// TwinCAT 3 PLC project ASRS
// ProgramVersion: 3.1.4024.0
// libraries:
//   Tc2_Standard, * (Beckhoff Automation GmbH)
//   Tc2_System, * (Beckhoff Automation GmbH)
//   Tc3_Module, * (Beckhoff Automation GmbH)
// project tree:
//   / Class Diagram.TcCD (not stored), Class Diagram_1.TcCD (not stored), PlcTask.TcTTO
//   DUTs/Enum/ E_ConveyorMode.TcDUT, E_DiverterState.TcDUT, E_CraneState.TcDUT, E_AisleMode.TcDUT, E_SlotStatus.TcDUT, E_WarehouseState.TcDUT
//   DUTs/Structure/ ST_Alarm.TcDUT, ST_Parcel.TcDUT, ST_StorageSlot.TcDUT, ST_Position.TcDUT, ST_CraneJob.TcDUT, ST_HMI_Search.TcDUT (not stored)
//   GVLs/ GVL_IO.TcGVL, GVL_Config.TcGVL, GVL_Warehouse.TcGVL
//   POUs/ITFs/ I_Conveyor.TcIO, I_Diverter.TcIO, I_Crane.TcIO
//   POUs/Entity/ FB_Conveyor.TcPOU, FB_BiDirectionConveyor.TcPOU, FB_RAT.TcPOU, FB_Crane.TcPOU
//   POUs/Controller/ FB_InFeedController.TcPOU, FB_LoopController.TcPOU, FB_AisleController.TcPOU, FB_CraneController.TcPOU, FB_OutFeedController.TcPOU
//   POUs/ FB_WareHouseController.TcPOU, MAIN.TcPOU
// real-time tasks:
//   TASK PlcTask: cycle T#10ms, priority 20, ADS port 350
//   TASK PlcTask1: cycle T#10ms, priority 21, ADS port 351

CONFIGURATION ASRS
    RESOURCE PLC ON TwinCAT3
        TASK PlcTask(INTERVAL := T#10ms, PRIORITY := 20);
        PROGRAM MAIN WITH PlcTask : MAIN;
    END_RESOURCE
END_CONFIGURATION

// ---- DUTs/Enum/E_ConveyorMode.TcDUT
{attribute 'qualified_only'}
{attribute 'strict'}

TYPE E_ConveyorMode :
(
    IDLE              := 0,
    RUNNING_FORWARD   := 1,
    RUNNING_BACKWARD  := 2,
    FAULT             := 3
);
END_TYPE

// ---- DUTs/Enum/E_DiverterState.TcDUT
{attribute 'qualified_only'}
{attribute 'strict'}
{attribute 'reflection'}
TYPE E_DiverterState :
(
    IDLE      := 0,
    LIFTING   := 10,
    DIVERTING := 20,
    LOWERING  := 30,
	DONE := 40,
    FAULT     := 90
);
END_TYPE

// ---- DUTs/Enum/E_CraneState.TcDUT
{attribute 'qualified_only'}
{attribute 'strict'}
TYPE E_CraneState :
(
    IDLE            := 0,
    MOVING_TO_PICK  := 10,
	READY_TO_PICK   := 15,
    PICKING         := 20,
	READY_TO_MOVE   := 25,
    MOVING_TO_PLACE := 30,
    PLACING         := 40,
    RETURNING_HOME  := 50,
    FAULT           := 99
);
END_TYPE

// ---- DUTs/Enum/E_AisleMode.TcDUT
{attribute 'qualified_only'}
{attribute 'strict'}
TYPE E_AisleMode :
(
    IDLE                := 0,
    RECEIVING_FROM_LOOP := 10,
    TRANSPORT_TO_CRANE  := 20,
    WAITING_FOR_PICK    := 30,
    READY_FOR_DROP      := 40,
    TRANSPORT_TO_LOOP   := 50,
    FAULT               := 99
);
END_TYPE

// ---- DUTs/Enum/E_SlotStatus.TcDUT
{attribute 'qualified_only'}
{attribute 'strict'}
TYPE E_SlotStatus :
(
    EMPTY        := 0,
    RESERVED_IN  := 1,
    OCCUPIED     := 2,
    RESERVED_OUT := 3,
    BLOCKED      := 4
);
END_TYPE

// ---- DUTs/Enum/E_WarehouseState.TcDUT
{attribute 'qualified_only'}
{attribute 'strict'}
TYPE E_WarehouseState :
(
    IDLE    := 0,
    RUNNING := 1,
    PAUSED  := 2,
    FAULT   := 99
);
END_TYPE

// ---- DUTs/Structure/ST_Alarm.TcDUT
TYPE ST_Alarm :
STRUCT
	bActive     : BOOL;
    sSource     : STRING(50);
    sMessage    : STRING(100);
END_STRUCT
END_TYPE

// ---- DUTs/Structure/ST_Parcel.TcDUT
TYPE ST_Parcel :
STRUCT
    sID          : STRING(20);
    sDescription : STRING(40);
    fWeight      : REAL;
    nTargetAisle : INT;
    bIsHeavy     : BOOL;
END_STRUCT
END_TYPE

// ---- DUTs/Structure/ST_StorageSlot.TcDUT
TYPE ST_StorageSlot :
STRUCT
    eStatus      : E_SlotStatus;
    stParcel     : ST_Parcel;
    bIsRear      : BOOL;
    bMaintenance : BOOL;
END_STRUCT
END_TYPE

// ---- DUTs/Structure/ST_Position.TcDUT
TYPE ST_Position :
STRUCT
    nCol            : INT;
    nRow            : INT;
    fTargetX        : LREAL;
    fTargetY        : LREAL;
    bIsAisleStation : BOOL;
END_STRUCT
END_TYPE

// ---- DUTs/Structure/ST_CraneJob.TcDUT
TYPE ST_CraneJob :
STRUCT
    bValid    : BOOL;
    bIsStore  : BOOL;
    nAisle    : INT;
    stRackPos : ST_Position;
    stParcel  : ST_Parcel;
END_STRUCT
END_TYPE

// ---- GVLs/GVL_IO.TcGVL
{attribute 'qualified_only'}
VAR_GLOBAL
	

	bParcelReady            : BOOL;
	bOutfeedReq             : BOOL;
    // Infeed conveyor
    bInfeedSensor           : BOOL;
    bInfeedBlocker          : BOOL;
    bInfeedMotor            : BOOL;

    // Infeed RAT (transfers parcel from infeed conveyor onto loop)
    bInfeedRatSensor        : BOOL;
    bInfeedRatLift          : BOOL;
    bInfeedRatTravel        : BOOL;
    bInfeedRatUp            : BOOL;
    bInfeedRatDown          : BOOL;

    // Main loop conveyor
    bLoopMotor              : BOOL;
    bLoopSensor             : BOOL;
	bLoopParcelMainBlocker  : BOOL;
    // Aisle 1 junction on loop
    bAisle1ApproachSensor   : BOOL;
    bAisle1StopBlocker      : BOOL;
    bAisle1RatLift          : BOOL;
    bAisle1RatTravel        : BOOL;
    bRat1Sensor             : BOOL;
    bRat1Up                 : BOOL;
    bRat1Down               : BOOL;

    // Aisle 2 junction on loop
    bAisle2ApproachSensor   : BOOL;
    bAisle2StopBlocker      : BOOL;
    bAisle2RatLift          : BOOL;
    bAisle2RatTravel        : BOOL;
    bRat2Sensor             : BOOL;
    bRat2Up                 : BOOL;
    bRat2Down               : BOOL;

    // Outfeed junction on loop
    bOutfeedApproachSensor  : BOOL;
	bOutfeedExitSensor      : BOOL;
    bOutfeedStopBlocker     : BOOL;
    bOutfeedRatLift         : BOOL;
    bOutfeedRatTravel       : BOOL;
    bOutfeedRatSensor       : BOOL;
    bOutfeedRatUp           : BOOL;
    bOutfeedRatDown         : BOOL;

    // Aisle 1 conveyor
    bAisle1EntrySensor      : BOOL;
    bAisle1CraneStation     : BOOL;
    bAisle1MotorForward     : BOOL;
    bAisle1MotorReverse     : BOOL;

    // Aisle 2 conveyor
    bAisle2EntrySensor      : BOOL;
    bAisle2CraneStation     : BOOL;
    bAisle2MotorForward     : BOOL;
    bAisle2MotorReverse     : BOOL;

    // Outfeed conveyor
    bOutfeedSensor          : BOOL;
    bOutfeedMotor           : BOOL;

    // Crane 1
    fCrane1PosX             : LREAL;
    fCrane1PosY             : LREAL;
    bCrane1ForksExtended    : BOOL;
    bCrane1ForksHome        : BOOL;
    bCrane1MotorX           : BOOL;
    bCrane1MotorY           : BOOL;
    bCrane1ForksOut         : BOOL;
    bCrane1EStop            : BOOL;
	bCrane1pick             : BOOL;
	bCrane1drop             : BOOL;
    // Crane 2
    fCrane2PosX             : LREAL;
    fCrane2PosY             : LREAL;
    bCrane2ForksExtended    : BOOL;
    bCrane2ForksHome        : BOOL;
    bCrane2MotorX           : BOOL;
    bCrane2MotorY           : BOOL;
    bCrane2ForksOut         : BOOL;
    bCrane2EStop            : BOOL;
	bCrane2pick				: BOOL;
	bCrane2drop             : BOOL;
END_VAR

// ---- GVLs/GVL_Config.TcGVL
{attribute 'qualified_only'}
VAR_GLOBAL CONSTANT
    MAX_COLUMNS         : INT := 10;
    MAX_ROWS            : INT := 4;
	
	HEAVY_RACK_STARTING_ROW : INT := 3;
	
    WEIGHT_LIMIT_HEAVY  : REAL := 100.0;

    COLUMN_SPACING      : LREAL := 1200.0;
    ROW_SPACING         : LREAL := 800.0;
    HOME_X              : LREAL := 0.0;
    HOME_Y              : LREAL := 0.0;

    T_RAT_LIFT_TIMEOUT  : TIME := T#4S;
    T_CRANE_MOVE_TIMEOUT: TIME := T#60S;
    T_FORK_TIMEOUT      : TIME := T#8S;
    T_JAM_TIMEOUT       : TIME := T#10S;

    CRANE_POS_TOLERANCE : LREAL := 5.0;
    CRANE1_AISLE        : INT   := 1;
    CRANE2_AISLE        : INT   := 2;
END_VAR

// ---- GVLs/GVL_Warehouse.TcGVL
{attribute 'qualified_only'}
VAR_GLOBAL PERSISTENT
    arrRack              : ARRAY[1..GVL_Config.MAX_ROWS, 1..GVL_Config.MAX_COLUMNS] OF ST_StorageSlot;
    nTotalStoredCount    : UDINT;
    nTotalRetrievedCount : UDINT;
    sWarehouseName       : STRING := 'IntimeTec_ASRS_01';
    bRackInitialized     : BOOL;
END_VAR

VAR_GLOBAL
    bSystemAutoMode      : BOOL := FALSE;
    bEmergencyStop       : BOOL := FALSE;
    sSystemStatusMsg     : STRING(80) := 'System Ready';
    stHmiSearch          : ST_HMI_Search;
	bStartRetrieval      : BOOL;
	bRetrievalRow        : INT;
	bRetrievalCol        : INT;
	
	bAlarmActive         : BOOL;
    sAlarmMessage        : STRING;
    arrAlarms            : ARRAY[1..10] OF ST_Alarm;
    nAlarmCount          : INT;
END_VAR

// ---- POUs/ITFs/I_Conveyor.TcIO
INTERFACE I_Conveyor

PROPERTY eMode : E_ConveyorMode
GET
END_GET
END_PROPERTY

PROPERTY fCurrentSpeed : LREAL
GET
END_GET
SET
END_SET
END_PROPERTY

METHOD M_Reset : BOOL
VAR_INPUT
END_VAR
END_METHOD

METHOD M_Run : BOOL
VAR_INPUT
	bForward : BOOL;
END_VAR
END_METHOD

METHOD M_Stop : BOOL
VAR_INPUT
END_VAR
END_METHOD

END_INTERFACE

// ---- POUs/ITFs/I_Diverter.TcIO
INTERFACE I_Diverter

PROPERTY bError : BOOL
GET
END_GET
END_PROPERTY

PROPERTY bLiftUp : BOOL
GET
END_GET
END_PROPERTY

PROPERTY bTravelMotorRun : BOOL
GET
END_GET
END_PROPERTY

PROPERTY eState : E_DiverterState
GET
END_GET
END_PROPERTY

METHOD M_Divert
VAR_INPUT
END_VAR
END_METHOD

METHOD M_Stop
VAR_INPUT
END_VAR
END_METHOD

END_INTERFACE

// ---- POUs/ITFs/I_Crane.TcIO
INTERFACE I_Crane

PROPERTY bBusy : BOOL
GET
END_GET
END_PROPERTY

PROPERTY bError : BOOL
GET
END_GET
END_PROPERTY

PROPERTY eState : E_CraneState
GET
END_GET
END_PROPERTY

METHOD M_Reset
VAR_INPUT
END_VAR
END_METHOD

METHOD M_StartJob
VAR_INPUT
    stPick  : ST_Position;
    stPlace : ST_Position;
END_VAR
END_METHOD

END_INTERFACE

// ---- POUs/MAIN.TcPOU
PROGRAM MAIN
VAR
    fbWarehouse : FB_WareHouseController;
    bFirstScan  : BOOL := TRUE;
	bStart      : BOOL;
END_VAR

IF bFirstScan THEN
    GVL_Warehouse.bSystemAutoMode := FALSE;
    GVL_Warehouse.bEmergencyStop  := FALSE;
    IF NOT GVL_Warehouse.bRackInitialized THEN
        fbWarehouse.M_InitRack();
    END_IF
    bFirstScan := FALSE;
END_IF

IF bStart AND NOT GVL_Warehouse.bEmergencyStop  THEN
	fbWarehouse();
	GVL_Warehouse.sSystemStatusMsg:= 'System Operating';
ELSE
	GVL_Warehouse.sSystemStatusMsg:= 'System Stopped';
END_IF

END_PROGRAM

// ---- POUs/FB_WareHouseController.TcPOU
FUNCTION_BLOCK FB_WareHouseController
VAR_OUTPUT
    bError  : BOOL;
    eState  : E_WarehouseState := E_WarehouseState.IDLE;
END_VAR
VAR
   
    fbInfeedBelt    : FB_Conveyor;
    fbLoopBelt      : FB_Conveyor;
    fbAisle1Belt    : FB_BiDirectionConveyor;
    fbAisle2Belt    : FB_BiDirectionConveyor;
    fbOutfeedBelt   : FB_Conveyor;
    fbInfeedRat     : FB_RAT;
    fbAisle1Rat     : FB_RAT;
    fbAisle2Rat     : FB_RAT;
    fbOutfeedRat    : FB_RAT;
    fbCrane1        : FB_Crane;
    fbCrane2        : FB_Crane;

    
    fbInfeed        : FB_InFeedController;
    fbLoop          : FB_LoopController;
    fbAisle1        : FB_AisleController;
    fbAisle2        : FB_AisleController;
    fbCraneCtrl1    : FB_CraneController;
    fbCraneCtrl2    : FB_CraneController;
    fbOutfeed       : FB_OutFeedController;

    
    arrJobs         : ARRAY[1..20] OF ST_CraneJob;
    nHead           : INT := 1;
    nTail           : INT := 1;
    nCount          : INT := 0;

    nTargetAisle    : INT := 0;
    
	bAisle1RetrievalPending : BOOL;   
	bAisle2RetrievalPending : BOOL; 
	bReset: BOOL;
END_VAR


fbInfeedBelt();
fbLoopBelt();

fbAisle1Belt(
    bEntrySensor        := GVL_IO.bAisle1EntrySensor,
    bCraneStationSensor := GVL_IO.bAisle1CraneStation
);
fbAisle2Belt(
    bEntrySensor        := GVL_IO.bAisle2EntrySensor,
    bCraneStationSensor := GVL_IO.bAisle2CraneStation
);
fbOutfeedBelt();

fbInfeedRat(
    bSensorOccupied := GVL_IO.bInfeedRatSensor,
    bSensorIsUp     := GVL_IO.bInfeedRatUp,
    bSensorIsDown   := GVL_IO.bInfeedRatDown
);
fbAisle1Rat(
    bSensorOccupied := GVL_IO.bRat1Sensor,
    bSensorIsUp     := GVL_IO.bRat1Up,
    bSensorIsDown   := GVL_IO.bRat1Down
);
fbAisle2Rat(
    bSensorOccupied := GVL_IO.bRat2Sensor,
    bSensorIsUp     := GVL_IO.bRat2Up,
    bSensorIsDown   := GVL_IO.bRat2Down
);
fbOutfeedRat(
    bSensorOccupied := GVL_IO.bOutfeedRatSensor,
    bSensorIsUp     := GVL_IO.bOutfeedRatUp,
    bSensorIsDown   := GVL_IO.bOutfeedRatDown
);

fbCrane1(
    fPosX          := GVL_IO.fCrane1PosX,
    fPosY          := GVL_IO.fCrane1PosY,
    bForksHome     := GVL_IO.bCrane1ForksHome
);
fbCrane2(
    fPosX          := GVL_IO.fCrane2PosX,
    fPosY          := GVL_IO.fCrane2PosY,
    bForksHome     := GVL_IO.bCrane2ForksHome 
);


GVL_IO.bCrane1MotorX  := fbCrane1.bMotorX;
GVL_IO.bCrane1MotorY  := fbCrane1.bMotorY;
GVL_IO.bCrane1ForksOut:= fbCrane1.bForksOut;
GVL_IO.bCrane2MotorX  := fbCrane2.bMotorX;
GVL_IO.bCrane2MotorY  := fbCrane2.bMotorY;
GVL_IO.bCrane2ForksOut:= fbCrane2.bForksOut;
GVL_IO.bCrane2ForksExtended  := fbCrane2.bForksExtended;
GVL_IO.bCrane1ForksExtended :=  fbCrane1.bForksExtended  ;



IF GVL_Warehouse.bEmergencyStop THEN
    eState := E_WarehouseState.FAULT;
END_IF

IF eState = E_WarehouseState.FAULT THEN
    bError := TRUE;
    RETURN;
END_IF


fbInfeed(iInfeedBelt := fbInfeedBelt, iInfeedRat := fbInfeedRat);

fbLoop(
    nTargetAisle    := nTargetAisle,
    bOutfeedRequest := GVL_IO.bOutfeedReq,
    iLoopBelt       := fbLoopBelt,
    iAisle1Rat      := fbAisle1Rat,
    iAisle2Rat      := fbAisle2Rat,
    iOutfeedRat     := fbOutfeedRat
);

fbAisle1(
    nAisleNumber    := 1,
    bInboundRequest := (nTargetAisle = 1) AND fbLoop.bLoopReady = FALSE,
    bOutboundRequest:= bAisle1RetrievalPending,                 
    bCranePickDone  := GVL_IO.bCrane1pick,
    bCraneDropDone  := GVL_IO.bCrane1drop,
    iAisleBelt      := fbAisle1Belt
);

fbAisle2(
    nAisleNumber    := 2,
    bInboundRequest := (nTargetAisle = 2) AND fbLoop.bLoopReady = FALSE,
    bOutboundRequest:= bAisle2RetrievalPending,                  
    bCranePickDone  := GVL_IO.bCrane2pick,
    bCraneDropDone  := GVL_IO.bCrane2drop,
    iAisleBelt      := fbAisle2Belt
);

fbCraneCtrl1(nAisleNumber := 1, iCrane := fbCrane1);
fbCraneCtrl2(nAisleNumber := 2, iCrane := fbCrane2);

fbOutfeed(iOutfeedBelt := fbOutfeedBelt);


IF GVL_IO.bParcelReady THEN
    M_RouteParcel();
END_IF

IF GVL_IO.bCrane1drop THEN
    GVL_IO.bCrane1drop := FALSE;
    nTargetAisle := 0;
    bAisle1RetrievalPending := FALSE;   
END_IF
IF GVL_IO.bCrane2drop THEN
    GVL_IO.bCrane2drop := FALSE;
    nTargetAisle := 0;
    bAisle2RetrievalPending := FALSE;   
END_IF

IF GVL_IO.bCrane1pick THEN
    GVL_IO.bCrane1pick := FALSE;
    nTargetAisle := 0;   
END_IF
IF GVL_IO.bCrane2pick THEN
    GVL_IO.bCrane2pick := FALSE;
    nTargetAisle := 0;
END_IF

IF GVL_Warehouse.bStartRetrieval THEN
	M_RequestRetrieval(GVL_Warehouse.bRetrievalCol, GVL_Warehouse.bRetrievalRow);
	GVL_Warehouse.bStartRetrieval := FALSE;
	GVL_Warehouse.bRetrievalRow := 0;
	GVL_Warehouse.bRetrievalCol := 0;
	
END_IF

IF fbAisle1.eMode = E_AisleMode.IDLE  AND fbAisle2.eMode = E_AisleMode.IDLE  THEN
	GVL_IO.bLoopParcelMainBlocker := FALSE;
ELSE
	GVL_IO.bLoopParcelMainBlocker := TRUE;
END_IF

M_DispatchJobs();


IF GVL_Warehouse.stHmiSearch.bTriggerSearch THEN
    M_HmiSearch();
END_IF


bError := fbInfeed.bError OR fbLoop.bError OR fbAisle1.bError OR fbAisle2.bError
          OR fbCraneCtrl1.bError OR fbCraneCtrl2.bError OR fbOutfeed.bError;


M_UpdateAlarms();

METHOD PRIVATE M_DispatchJobs
VAR
    stJob : ST_CraneJob;
	stEmptySlot : ST_StorageSlot;
END_VAR
IF nCount = 0 THEN RETURN; END_IF

stJob := arrJobs[nHead];
IF stJob.bIsStore THEN
	IF stJob.nAisle = 1 AND NOT fbCraneCtrl1.bBusy THEN
		IF fbCraneCtrl1.M_AssignStore(stJob := stJob) THEN
			GVL_Warehouse.arrRack[stJob.stRackPos.nRow, stJob.stRackPos.nCol].eStatus := E_SlotStatus.RESERVED_IN;
			arrJobs[nHead].bValid := FALSE;
			nHead  := nHead MOD 20 + 1;
			nCount := nCount - 1;
		END_IF
	ELSIF stJob.nAisle = 2 AND NOT fbCraneCtrl2.bBusy THEN
		IF fbCraneCtrl2.M_AssignStore(stJob := stJob) THEN
			GVL_Warehouse.arrRack[stJob.stRackPos.nRow, stJob.stRackPos.nCol].eStatus := E_SlotStatus.RESERVED_IN;
			arrJobs[nHead].bValid := FALSE;
			nHead  := nHead MOD 20 + 1;
			nCount := nCount - 1;
		END_IF
	END_IF
ELSE
	IF stJob.nAisle = 1 AND NOT fbCraneCtrl1.bBusy THEN
		IF fbCraneCtrl1.M_AssignRetrieve(stJob := stJob) THEN
			GVL_Warehouse.arrRack[stJob.stRackPos.nRow, stJob.stRackPos.nCol].eStatus := E_SlotStatus.RESERVED_OUT;
			arrJobs[nHead].bValid := FALSE;
			nHead  := nHead MOD 20 + 1;
			nCount := nCount - 1;
		END_IF
	ELSIF stJob.nAisle = 2 AND NOT fbCraneCtrl2.bBusy THEN
		IF fbCraneCtrl2.M_AssignRetrieve(stJob := stJob) THEN
			GVL_Warehouse.arrRack[stJob.stRackPos.nRow, stJob.stRackPos.nCol].eStatus := E_SlotStatus.RESERVED_OUT;
			arrJobs[nHead].bValid := FALSE;
			nHead  := nHead MOD 20 + 1;
			nCount := nCount - 1;
		END_IF
	END_IF
END_IF
END_METHOD

METHOD PRIVATE M_Enqueue
VAR_INPUT
    stJob : ST_CraneJob;
END_VAR
IF nCount >= 20 THEN 
	RETURN; 
END_IF
arrJobs[nTail] := stJob;
nTail  := nTail MOD 20 + 1;
nCount := nCount + 1;
END_METHOD

METHOD PRIVATE M_HmiSearch
VAR
    nCol : INT;
    nRow : INT;
END_VAR
GVL_Warehouse.stHmiSearch.bMatchFound := FALSE;
FOR nRow := 1 TO GVL_Config.MAX_ROWS DO
    FOR nCol := 1 TO GVL_Config.MAX_COLUMNS DO
        IF GVL_Warehouse.arrRack[ nRow, nCol ].eStatus = E_SlotStatus.OCCUPIED AND
           GVL_Warehouse.arrRack[ nRow, nCol ].stParcel.sID = GVL_Warehouse.stHmiSearch.sSearchID THEN
            GVL_Warehouse.stHmiSearch.bMatchFound      := TRUE;
            GVL_Warehouse.stHmiSearch.nFoundCol        := nCol;
            GVL_Warehouse.stHmiSearch.nFoundRow        := nRow;
            GVL_Warehouse.stHmiSearch.stSelectedParcel := GVL_Warehouse.arrRack[ nRow, nCol ].stParcel;
            GVL_Warehouse.stHmiSearch.eSelectedStatus  := GVL_Warehouse.arrRack[ nRow, nCol ].eStatus;
        END_IF
    END_FOR
END_FOR
GVL_Warehouse.stHmiSearch.bTriggerSearch := FALSE;
END_METHOD

METHOD M_InitRack
VAR
    nCol : INT;
    nRow : INT;
END_VAR
FOR nRow := 1 TO GVL_Config.MAX_ROWS DO
    FOR nCol := 1 TO GVL_Config.MAX_COLUMNS DO
        GVL_Warehouse.arrRack[nRow, nCol].eStatus     := E_SlotStatus.EMPTY;
        GVL_Warehouse.arrRack[nRow, nCol].bMaintenance:= FALSE;
        GVL_Warehouse.arrRack[nRow, nCol].bIsRear     := (nRow MOD 2 = 0);
    END_FOR
END_FOR
GVL_Warehouse.bRackInitialized := TRUE;
END_METHOD

METHOD M_RequestRetrieval : BOOL
VAR_INPUT
    nCol : INT;
    nRow : INT;
END_VAR
VAR
    stJob : ST_CraneJob;
END_VAR
IF nCol < 1 OR nCol > GVL_Config.MAX_COLUMNS OR
   nRow < 1 OR nRow > GVL_Config.MAX_ROWS THEN
    M_RequestRetrieval := FALSE;
    RETURN;
END_IF

IF GVL_Warehouse.arrRack[nRow, nCol].eStatus <> E_SlotStatus.OCCUPIED THEN
    M_RequestRetrieval := FALSE;
    RETURN;
END_IF

GVL_Warehouse.arrRack[nRow, nCol].eStatus := E_SlotStatus.RESERVED_OUT;

stJob.bValid             := TRUE;
stJob.bIsStore           := FALSE;
stJob.stParcel           := GVL_Warehouse.arrRack[nRow, nCol].stParcel;
stJob.stRackPos.nCol     := nCol;
stJob.stRackPos.nRow     := nRow;
stJob.stRackPos.fTargetX := (nCol - 1) * GVL_Config.COLUMN_SPACING;
stJob.stRackPos.fTargetY := (nRow - 1) * GVL_Config.ROW_SPACING;
stJob.nAisle             := SEL(stJob.stParcel.bIsHeavy, GVL_Config.CRANE1_AISLE, GVL_Config.CRANE2_AISLE);

M_Enqueue(stJob);



IF stJob.nAisle = 1 THEN
    bAisle1RetrievalPending := TRUE;
ELSIF stJob.nAisle = 2 THEN
    bAisle2RetrievalPending := TRUE;
END_IF
GVL_IO.bOutfeedReq := TRUE;
M_RequestRetrieval := TRUE;
END_METHOD

METHOD PRIVATE M_RouteParcel
VAR
    stJob  : ST_CraneJob;
    nCol   : INT;
    nRow   : INT;
    bFound : BOOL;
	nDecideRow : INT;
	nDecideCol : INT;
END_VAR

IF nTargetAisle = 0 THEN
    IF fbInfeed.stParcel.fWeight > 100 THEN
        nTargetAisle := GVL_Config.CRANE2_AISLE;
		nDecideRow := GVL_Config.HEAVY_RACK_STARTING_ROW;
    ELSE
        nTargetAisle := GVL_Config.CRANE1_AISLE;
		nDecideRow := 1;
    END_IF
ELSE
   
    GVL_IO.bInfeedBlocker := TRUE;
    RETURN;   
END_IF


bFound := FALSE;



FOR nRow := nDecideRow TO GVL_Config.MAX_ROWS DO
    FOR nCol := 1 TO GVL_Config.MAX_COLUMNS DO
        IF GVL_Warehouse.arrRack[nRow, nCol].bIsRear
            AND GVL_Warehouse.arrRack[nRow, nCol].eStatus = E_SlotStatus.EMPTY
            AND NOT GVL_Warehouse.arrRack[nRow, nCol].bMaintenance THEN
            bFound := TRUE;
            EXIT;
        END_IF
    END_FOR
    IF bFound THEN
		EXIT; 
	END_IF
END_FOR


IF NOT bFound THEN
    FOR nRow := nDecideRow TO GVL_Config.MAX_ROWS DO
    	FOR nCol := 1 TO GVL_Config.MAX_COLUMNS DO
        	IF NOT GVL_Warehouse.arrRack[nRow, nCol].bIsRear
            	AND GVL_Warehouse.arrRack[nRow, nCol].eStatus = E_SlotStatus.EMPTY
            	AND NOT GVL_Warehouse.arrRack[nRow, nCol].bMaintenance THEN
            	bFound := TRUE;
            	EXIT;
        	END_IF
    	END_FOR
    	IF bFound THEN 
			EXIT; 
		END_IF
	END_FOR
END_IF

IF NOT bFound THEN
    GVL_Warehouse.sSystemStatusMsg := 'Rack full';
    RETURN;
END_IF

GVL_Warehouse.arrRack[nRow, nCol].eStatus  := E_SlotStatus.RESERVED_IN;
GVL_Warehouse.arrRack[nRow, nCol].stParcel := fbInfeed.stParcel;

stJob.bValid             := TRUE;
stJob.bIsStore           := TRUE;
stJob.nAisle             := nTargetAisle;
stJob.stParcel           := fbInfeed.stParcel;
stJob.stRackPos.nCol     := nCol;
stJob.stRackPos.nRow     := nRow;
stJob.stRackPos.fTargetX := (nCol - 1) * GVL_Config.COLUMN_SPACING;
stJob.stRackPos.fTargetY := (nRow - 1) * GVL_Config.ROW_SPACING;

M_Enqueue(stJob);
END_METHOD

METHOD M_UpdateAlarms : BOOL

VAR
	nCounter : INT;
END_VAR


IF bReset THEN
	FOR nCounter := 1 TO 10 DO
		GVL_Warehouse.arrAlarms[nCounter].bActive  := FALSE;
		GVL_Warehouse.arrAlarms[nCounter].sSource  := '';
		GVL_Warehouse.arrAlarms[nCounter].sMessage := '';
	END_FOR
	bReset := FALSE;
END_IF

IF GVL_Warehouse.nAlarmCount = 10 THEN
	RETURN;
END_IF

IF GVL_Warehouse.nAlarmCount = 0 THEN
	GVL_Warehouse.bAlarmActive := FALSE ;
    GVL_Warehouse.sAlarmMessage := 'No Fault. Working Properly';
ELSE
	GVL_Warehouse.bAlarmActive := TRUE ;
    GVL_Warehouse.sAlarmMessage := 'Error Occurred. See the Alarm Screen';
END_IF


IF fbInfeed.bError THEN
    GVL_Warehouse.nAlarmCount := GVL_Warehouse.nAlarmCount + 1;
    GVL_Warehouse.arrAlarms[GVL_Warehouse.nAlarmCount].bActive  := TRUE;
    GVL_Warehouse.arrAlarms[GVL_Warehouse.nAlarmCount].sSource  := 'InFeed';
    GVL_Warehouse.arrAlarms[GVL_Warehouse.nAlarmCount].sMessage := 'InFeed Controller Error';
END_IF

IF fbLoop.bError THEN
    GVL_Warehouse.nAlarmCount := GVL_Warehouse.nAlarmCount + 1;
    GVL_Warehouse.arrAlarms[GVL_Warehouse.nAlarmCount].bActive  := TRUE;
    GVL_Warehouse.arrAlarms[GVL_Warehouse.nAlarmCount].sSource  := 'Loop';
    GVL_Warehouse.arrAlarms[GVL_Warehouse.nAlarmCount].sMessage := 'Loop Controller Error';
END_IF

IF fbAisle1.bError THEN
    GVL_Warehouse.nAlarmCount := GVL_Warehouse.nAlarmCount + 1;
    GVL_Warehouse.arrAlarms[GVL_Warehouse.nAlarmCount].bActive  := TRUE;
    GVL_Warehouse.arrAlarms[GVL_Warehouse.nAlarmCount].sSource  := 'Aisle1';
    GVL_Warehouse.arrAlarms[GVL_Warehouse.nAlarmCount].sMessage := 'Aisle 1 Controller Error';
END_IF

IF fbAisle2.bError THEN
    GVL_Warehouse.nAlarmCount := GVL_Warehouse.nAlarmCount + 1;
    GVL_Warehouse.arrAlarms[GVL_Warehouse.nAlarmCount].bActive  := TRUE;
    GVL_Warehouse.arrAlarms[GVL_Warehouse.nAlarmCount].sSource  := 'Aisle2';
    GVL_Warehouse.arrAlarms[GVL_Warehouse.nAlarmCount].sMessage := 'Aisle 2 Controller Error';
END_IF

IF fbCraneCtrl1.bError THEN
    GVL_Warehouse.nAlarmCount := GVL_Warehouse.nAlarmCount + 1;
    GVL_Warehouse.arrAlarms[GVL_Warehouse.nAlarmCount].bActive  := TRUE;
    GVL_Warehouse.arrAlarms[GVL_Warehouse.nAlarmCount].sSource  := 'Crane1';
    GVL_Warehouse.arrAlarms[GVL_Warehouse.nAlarmCount].sMessage := 'Crane 1 Controller Error';
END_IF

IF fbCraneCtrl2.bError THEN
    GVL_Warehouse.nAlarmCount := GVL_Warehouse.nAlarmCount + 1;
    GVL_Warehouse.arrAlarms[GVL_Warehouse.nAlarmCount].bActive  := TRUE;
    GVL_Warehouse.arrAlarms[GVL_Warehouse.nAlarmCount].sSource  := 'Crane2';
    GVL_Warehouse.arrAlarms[GVL_Warehouse.nAlarmCount].sMessage := 'Crane 2 Controller Error';
END_IF

IF fbOutfeed.bError THEN
    GVL_Warehouse.nAlarmCount := GVL_Warehouse.nAlarmCount + 1;
    GVL_Warehouse.arrAlarms[GVL_Warehouse.nAlarmCount].bActive  := TRUE;
    GVL_Warehouse.arrAlarms[GVL_Warehouse.nAlarmCount].sSource  := 'OutFeed';
    GVL_Warehouse.arrAlarms[GVL_Warehouse.nAlarmCount].sMessage := 'OutFeed Controller Error';
END_IF

IF GVL_Warehouse.bEmergencyStop THEN
    GVL_Warehouse.nAlarmCount := GVL_Warehouse.nAlarmCount + 1;
    GVL_Warehouse.arrAlarms[GVL_Warehouse.nAlarmCount].bActive  := TRUE;
    GVL_Warehouse.arrAlarms[GVL_Warehouse.nAlarmCount].sSource  := 'System';
    GVL_Warehouse.arrAlarms[GVL_Warehouse.nAlarmCount].sMessage := 'Emergency Stop Active';
END_IF
END_METHOD

END_FUNCTION_BLOCK

// ---- POUs/Entity/FB_Conveyor.TcPOU
FUNCTION_BLOCK FB_Conveyor IMPLEMENTS I_Conveyor
VAR_OUTPUT
    bConveyorError        : BOOL;
    bConveyorMotorRun     : BOOL;
    bConveyorMotorReverse : BOOL;
END_VAR
VAR
    eMode       : E_ConveyorMode := E_ConveyorMode.IDLE;
    fbJamTimer  : TON;
END_VAR


IF fbJamTimer.Q THEN
    eMode := E_ConveyorMode.FAULT;
END_IF

CASE eMode OF
    E_ConveyorMode.IDLE:
        bConveyorMotorRun     := FALSE;
        bConveyorMotorReverse := FALSE;

    E_ConveyorMode.RUNNING_FORWARD:
        bConveyorMotorRun     := TRUE;
        bConveyorMotorReverse := FALSE;

    E_ConveyorMode.RUNNING_BACKWARD:
        bConveyorMotorRun     := TRUE;
        bConveyorMotorReverse := TRUE;

    E_ConveyorMode.FAULT:
        bConveyorMotorRun     := FALSE;
        bConveyorMotorReverse := FALSE;
        bConveyorError        := TRUE;
END_CASE

PROPERTY bError : BOOL
GET
bError := bConveyorError;
END_GET
END_PROPERTY

PROPERTY bMotorReverse : BOOL
GET
bMotorReverse := bConveyorMotorReverse;
END_GET
END_PROPERTY

PROPERTY bMotorRun : BOOL
GET
bMotorRun := bConveyorMotorRun;
END_GET
END_PROPERTY

METHOD M_Reset
VAR_INPUT
END_VAR
bConveyorError := FALSE;
eMode  := E_ConveyorMode.IDLE;
END_METHOD

METHOD M_Run
VAR_INPUT
    bForward : BOOL;
END_VAR
IF eMode = E_ConveyorMode.FAULT THEN
	RETURN;
END_IF
IF bForward THEN
    eMode := E_ConveyorMode.RUNNING_FORWARD;
ELSE
    eMode := E_ConveyorMode.RUNNING_BACKWARD;
END_IF
END_METHOD

METHOD M_Stop
VAR_INPUT
END_VAR
eMode := E_ConveyorMode.IDLE;
END_METHOD

END_FUNCTION_BLOCK

// ---- POUs/Entity/FB_BiDirectionConveyor.TcPOU
FUNCTION_BLOCK FB_BiDirectionConveyor EXTENDS FB_Conveyor
VAR_INPUT
    bEntrySensor        : BOOL;
    bCraneStationSensor : BOOL;
END_VAR

SUPER^();

CASE eMode OF
    E_ConveyorMode.RUNNING_FORWARD:
        IF bCraneStationSensor THEN
            eMode := E_ConveyorMode.IDLE;
        END_IF

    E_ConveyorMode.RUNNING_BACKWARD:
        IF bEntrySensor THEN
            eMode := E_ConveyorMode.IDLE;
        END_IF
END_CASE

END_FUNCTION_BLOCK

// ---- POUs/Entity/FB_RAT.TcPOU
FUNCTION_BLOCK FB_RAT IMPLEMENTS I_Diverter
VAR_INPUT
    bSensorOccupied : BOOL;
    bSensorIsUp     : BOOL;
    bSensorIsDown   : BOOL;
END_VAR
VAR_OUTPUT
    bRatError          : BOOL;
    bIsLiftUp         : BOOL;
    bDivertMotorRun : BOOL;
END_VAR
VAR
    eRatState          : E_DiverterState := E_DiverterState.IDLE;
    fbLiftTimer     : TON;
    fbTravelTimer   : TON;
END_VAR


CASE eRatState OF
    E_DiverterState.IDLE:
        bIsLiftUp         := FALSE;
        bDivertMotorRun := FALSE;
		IF GVL_IO.bRat1Sensor THEN
           	
            GVL_IO.bAisle1StopBlocker := FALSE;
           
        END_IF

    E_DiverterState.LIFTING:
        bIsLiftUp := TRUE;
        IF bSensorIsUp THEN
            eRatState := E_DiverterState.DIVERTING;
        END_IF

    E_DiverterState.DIVERTING:
        bIsLiftUp         := TRUE;
        bDivertMotorRun := TRUE;
        IF NOT bSensorOccupied THEN
            eRatState := E_DiverterState.LOWERING;
        END_IF

    E_DiverterState.LOWERING:
        bIsLiftUp         := FALSE;
        bDivertMotorRun := FALSE;
        IF bSensorIsDown THEN
            eRatState := E_DiverterState.DONE;
        END_IF
	E_DiverterState.DONE:
		eRatState := E_DiverterState.IDLE;
		
    E_DiverterState.FAULT:
        bIsLiftUp         := FALSE;
        bDivertMotorRun := FALSE;
        bRatError          := TRUE;
END_CASE

PROPERTY bError : BOOL
GET
bError := bRatError;
END_GET
END_PROPERTY

PROPERTY bLiftUp : BOOL
GET
bLiftUp := bIsLiftUp;
END_GET
END_PROPERTY

PROPERTY bTravelMotorRun : BOOL
GET
bTravelMotorRun := bDivertMotorRun;
END_GET
END_PROPERTY

PROPERTY eState : E_DiverterState
GET
eState := eRatState;
END_GET
END_PROPERTY

METHOD M_Divert
VAR_INPUT
END_VAR
IF eRatState = E_DiverterState.IDLE THEN
    eRatState := E_DiverterState.LIFTING;
END_IF
END_METHOD

METHOD M_Stop
VAR_INPUT
END_VAR
bIsLiftUp         := FALSE;
bDivertMotorRun := FALSE;
eRatState          := E_DiverterState.IDLE;
END_METHOD

END_FUNCTION_BLOCK

// ---- POUs/Entity/FB_Crane.TcPOU
FUNCTION_BLOCK FB_Crane IMPLEMENTS I_Crane
VAR_INPUT
    fPosX           : LREAL;
    fPosY           : LREAL;
    bForksHome      : BOOL;
END_VAR
VAR_OUTPUT
    bCraneBusy           : BOOL;
    bCraneError          : BOOL;
    eCraneState          : E_CraneState := E_CraneState.IDLE;
    bMotorX         : BOOL;
    bMotorY         : BOOL;
    bForksOut       : BOOL;
	bForksExtended  : BOOL;
END_VAR
VAR
    stPickPos       : ST_Position;
    stPlacePos      : ST_Position;
	fbMoveTimer     : TON;
END_VAR


CASE eCraneState OF
    E_CraneState.IDLE:
        bCraneBusy    := FALSE;
        bMotorX  := FALSE;
        bMotorY  := FALSE;
        bForksOut:= FALSE;
		
    E_CraneState.MOVING_TO_PICK:
		bCraneBusy := TRUE;
		bMotorX    := TRUE;
		bMotorY    := TRUE;
		fbMoveTimer(IN := TRUE, PT := T#10S);
		IF fbMoveTimer.Q THEN
			fbMoveTimer(IN := FALSE);
			bMotorX     := FALSE;
			bMotorY     := FALSE;
			eCraneState := E_CraneState.READY_TO_PICK;
		END_IF
		
	E_CraneState.READY_TO_PICK:
	IF GVL_IO.bOutfeedReq OR GVL_IO.bAisle1CraneStation THEN
		eCraneState := E_CraneState.PICKING;
		bForksOut := TRUE;
		GVL_IO.bCrane1ForksHome := FALSE;
	END_IF
	
	
	
    E_CraneState.PICKING:
        bCraneBusy    := TRUE;
        IF bForksOut THEN
			IF bForksExtended THEN
					bForksOut := FALSE;
					bForksExtended := FALSE;
					eCraneState := E_CraneState.READY_TO_MOVE;
			END_IF
        END_IF
		
	 E_CraneState.READY_TO_MOVE:
		bCraneBusy     := TRUE;
        bForksExtended := FALSE;
		 IF bForksHome THEN
			 bForksOut := FALSE; 
			 eCraneState := E_CraneState.MOVING_TO_PLACE;
		 END_IF

    E_CraneState.MOVING_TO_PLACE:
       
            bMotorX := TRUE;
            bMotorY := TRUE;
			fbMoveTimer(IN := TRUE, PT := T#10S);
		IF fbMoveTimer.Q THEN    
			fbMoveTimer(IN := FALSE);  
			bMotorX := FALSE;
            bMotorY := FALSE;
            eCraneState  := E_CraneState.PLACING;
		END_IF      
       


    E_CraneState.PLACING:
        bCraneBusy    := TRUE;
        bForksOut:= TRUE;
        IF bForksExtended THEN
            bForksOut := FALSE;
			bForksExtended := FALSE;
            bCraneBusy     := FALSE;
            eCraneState    := E_CraneState.IDLE;
        END_IF

    E_CraneState.RETURNING_HOME:
        bCraneBusy   := TRUE;
        bMotorX := TRUE;
        bMotorY := TRUE;
        fbMoveTimer(IN := TRUE, PT := T#10S);
		IF fbMoveTimer.Q THEN
			fbMoveTimer(IN := FALSE);
			bMotorX := FALSE;
            bMotorY := FALSE;
            bCraneBusy   := FALSE;
            eCraneState  := E_CraneState.IDLE;
		END_IF

    E_CraneState.FAULT:
        bMotorX  := FALSE;
        bMotorY  := FALSE;
        bForksOut:= FALSE;
        bCraneBusy    := FALSE;
        bCraneError   := TRUE;
END_CASE

PROPERTY bBusy : BOOL
GET
bBusy := bCraneBusy;
END_GET
END_PROPERTY

PROPERTY bError : BOOL
GET
bError := bCraneError;
END_GET
END_PROPERTY

PROPERTY eState : E_CraneState
GET
eState := eCraneState;
END_GET
END_PROPERTY

METHOD M_Reset
VAR_INPUT
END_VAR
bCraneError := FALSE;
eCraneState := E_CraneState.RETURNING_HOME;
END_METHOD

METHOD M_StartJob 
VAR_INPUT
    stPick  : ST_Position;
    stPlace : ST_Position;
END_VAR
IF eCraneState <> E_CraneState.IDLE THEN
    RETURN;
END_IF
stPickPos  := stPick;
stPlacePos := stPlace;
eCraneState := E_CraneState.MOVING_TO_PICK;
END_METHOD

END_FUNCTION_BLOCK

// ---- POUs/Controller/FB_InFeedController.TcPOU
FUNCTION_BLOCK FB_InFeedController
VAR_OUTPUT
    bError          : BOOL;
    stParcel        : ST_Parcel;
END_VAR
VAR_INPUT
	iInfeedBelt     : I_Conveyor;
    iInfeedRat      : I_Diverter;
END_VAR
VAR
    nState : (IDLE, CONVEYING, WAIT_RAT_CLEAR, DONE) := IDLE;
END_VAR

// Write physical outputs
GVL_IO.bInfeedMotor   := iInfeedBelt.bMotorRun;
GVL_IO.bInfeedRatLift := iInfeedRat.bLiftUp;
GVL_IO.bInfeedRatTravel := iInfeedRat.bTravelMotorRun;

CASE nState OF

    IDLE:
        GVL_IO.bParcelReady := FALSE;
        
        IF GVL_IO.bInfeedSensor THEN
    
			IF NOT GVL_IO.bInfeedRatSensor THEN
				GVL_IO.bInfeedBlocker := FALSE;
			END_IF
			
            IF NOT GVL_IO.bInfeedBlocker THEN
                iInfeedBelt.M_Run(bForward := TRUE);
                nState := CONVEYING;
            END_IF
        END_IF

    CONVEYING:
        
        IF GVL_IO.bInfeedRatSensor THEN
			GVL_IO.bInfeedSensor := FALSE;
			GVL_IO.bInfeedBlocker := TRUE;
            iInfeedBelt.M_Stop();
            iInfeedRat.M_Divert();
            nState := WAIT_RAT_CLEAR;
			
        END_IF

    WAIT_RAT_CLEAR:
        
        IF NOT GVL_IO.bInfeedRatSensor THEN
			
            GVL_IO.bParcelReady := TRUE;
            nState := DONE;
        END_IF

    DONE:
       
		GVL_IO.bParcelReady := FALSE;
        nState := IDLE;

END_CASE

bError := iInfeedRat.bError OR iInfeedBelt.bError;

END_FUNCTION_BLOCK

// ---- POUs/Controller/FB_LoopController.TcPOU
FUNCTION_BLOCK FB_LoopController
VAR_INPUT
    nTargetAisle    : INT;
    bOutfeedRequest : BOOL;
	iLoopBelt       : I_Conveyor;
    iAisle1Rat      : I_Diverter;
    iAisle2Rat      : I_Diverter;
    iOutfeedRat     : I_Diverter;
END_VAR
VAR_OUTPUT
    bLoopReady      : BOOL;
    bError          : BOOL;
END_VAR

VAR
    nState : (MONITORING, DIVERT_A1, DIVERT_A2, DIVERT_OUT) := MONITORING;
END_VAR

// Write physical outputs
GVL_IO.bLoopMotor          := iLoopBelt.bMotorRun;
GVL_IO.bAisle1RatLift      := iAisle1Rat.bLiftUp;
GVL_IO.bAisle1RatTravel    := iAisle1Rat.bTravelMotorRun;
GVL_IO.bAisle2RatLift      := iAisle2Rat.bLiftUp;
GVL_IO.bAisle2RatTravel    := iAisle2Rat.bTravelMotorRun;
GVL_IO.bOutfeedRatLift     := iOutfeedRat.bLiftUp;
GVL_IO.bOutfeedRatTravel   := iOutfeedRat.bTravelMotorRun;


IF iAisle1Rat.eState = E_ConveyorMode.RUNNING_BACKWARD AND GVL_IO.bRat1Sensor THEN
	GVL_IO.bAisle1StopBlocker := FALSE;
END_IF
IF iAisle2Rat.eState = E_ConveyorMode.RUNNING_BACKWARD AND GVL_IO.bRat2Sensor THEN
	GVL_IO.bAisle2StopBlocker := FALSE;
END_IF


CASE nState OF

    MONITORING:
        bLoopReady := TRUE;
        iLoopBelt.M_Run(bForward := TRUE);
		
        // Parcel at Aisle 1 junction and Aisle 1 is the target
        IF GVL_IO.bAisle1ApproachSensor AND nTargetAisle = 1
            AND iAisle1Rat.eState = E_DiverterState.IDLE THEN
			GVL_IO.bLoopParcelMainBlocker := FALSE;
            GVL_IO.bAisle1StopBlocker := TRUE;
            nState := DIVERT_A1;

        // Parcel at Aisle 2 junction and Aisle 2 is the target
        ELSIF GVL_IO.bAisle2ApproachSensor AND nTargetAisle = 2
            AND iAisle2Rat.eState = E_DiverterState.IDLE THEN
			GVL_IO.bLoopParcelMainBlocker := FALSE;
            GVL_IO.bAisle2StopBlocker := TRUE;
            nState := DIVERT_A2;

        // Parcel at outfeed junction
        ELSIF GVL_IO.bOutfeedApproachSensor
            AND iOutfeedRat.eState = E_DiverterState.IDLE THEN
            GVL_IO.bOutfeedStopBlocker := TRUE;
            nState := DIVERT_OUT;
        END_IF

    DIVERT_A1:
        bLoopReady := FALSE;
        // Parcel centered on RAT sensor - execute divert
        IF GVL_IO.bRat1Sensor THEN
            iLoopBelt.M_Stop();
            GVL_IO.bAisle1StopBlocker := FALSE;
            iAisle1Rat.M_Divert();
        END_IF
        IF NOT GVL_IO.bAisle1EntrySensor AND iAisle1Rat.eState = E_DiverterState.IDLE AND NOT GVL_IO.bRat1Sensor THEN
			iAisle1Rat.M_Stop();
            nState := MONITORING;
        END_IF

    DIVERT_A2:
        bLoopReady := FALSE;
        IF GVL_IO.bRat2Sensor THEN
            iLoopBelt.M_Stop();
            GVL_IO.bAisle2StopBlocker := FALSE;
            iAisle2Rat.M_Divert();
        END_IF
        IF NOT GVL_IO.bAisle2EntrySensor AND iAisle2Rat.eState = E_DiverterState.IDLE AND NOT GVL_IO.bRat2Sensor THEN
			iAisle2Rat.M_Stop();
            nState := MONITORING;
        END_IF

    DIVERT_OUT:
        bLoopReady := FALSE;
        IF GVL_IO.bOutfeedRatSensor THEN
            iLoopBelt.M_Stop();
            GVL_IO.bOutfeedStopBlocker := FALSE;
            iOutfeedRat.M_Divert();
        END_IF
        IF GVL_IO.bOutfeedExitSensor AND  iOutfeedRat.eState = E_DiverterState.IDLE AND NOT GVL_IO.bOutfeedRatSensor THEN
            nState := MONITORING;
        END_IF

END_CASE

bError := iLoopBelt.bError OR iAisle1Rat.bError OR iAisle2Rat.bError OR iOutfeedRat.bError;

END_FUNCTION_BLOCK

// ---- POUs/Controller/FB_AisleController.TcPOU
FUNCTION_BLOCK FB_AisleController
VAR_INPUT
    nAisleNumber        : INT;
    bInboundRequest     : BOOL;
    bOutboundRequest    : BOOL;
    bCranePickDone      : BOOL;
    bCraneDropDone      : BOOL;
	iAisleBelt          : I_Conveyor;
END_VAR
VAR_OUTPUT
    bBoxAtPickPoint     : BOOL;
    bReadyForRetrieval  : BOOL;
    bError              : BOOL;
	eMode               : E_AisleMode := E_AisleMode.IDLE;
END_VAR

VAR
    
    bEntrySensor        : BOOL;
    bCraneStation       : BOOL;
END_VAR


ACT_ConfigureAisle();
CASE eMode OF

    E_AisleMode.IDLE:
        bBoxAtPickPoint    := FALSE;
        bReadyForRetrieval := FALSE;
        IF bInboundRequest THEN
            iAisleBelt.M_Run(bForward := TRUE);
            eMode := E_AisleMode.RECEIVING_FROM_LOOP;
        ELSIF bOutboundRequest THEN
            eMode := E_AisleMode.READY_FOR_DROP;
        END_IF

    E_AisleMode.RECEIVING_FROM_LOOP:
       
        IF bCraneStation THEN
			GVL_IO.bAisle1ApproachSensor := FALSE;
            iAisleBelt.M_Stop();
            bBoxAtPickPoint := TRUE;
            eMode := E_AisleMode.WAITING_FOR_PICK;
        ELSIF bEntrySensor AND NOT bCraneStation THEN
            eMode := E_AisleMode.TRANSPORT_TO_CRANE;
        END_IF

    E_AisleMode.TRANSPORT_TO_CRANE:
        iAisleBelt.M_Run(bForward := TRUE);
        IF bCraneStation THEN
            iAisleBelt.M_Stop();
            bBoxAtPickPoint := TRUE;
            eMode := E_AisleMode.WAITING_FOR_PICK;
        END_IF

    E_AisleMode.WAITING_FOR_PICK:
    IF bCranePickDone THEN
        bBoxAtPickPoint := FALSE;
        IF nAisleNumber = 1 THEN
            GVL_IO.bAisle1EntrySensor  := FALSE;
            GVL_IO.bAisle1CraneStation := FALSE;
        ELSE
            GVL_IO.bAisle2EntrySensor  := FALSE;
            GVL_IO.bAisle2CraneStation := FALSE;
        END_IF
        eMode := E_AisleMode.IDLE;
    END_IF

    E_AisleMode.READY_FOR_DROP:
       
        bReadyForRetrieval := TRUE;
        IF bCraneDropDone AND bCraneStation THEN
            bReadyForRetrieval := FALSE;
            iAisleBelt.M_Run(bForward := FALSE);
            eMode := E_AisleMode.TRANSPORT_TO_LOOP;
        END_IF

    E_AisleMode.TRANSPORT_TO_LOOP:
        
        IF bEntrySensor THEN
            iAisleBelt.M_Stop();
            eMode := E_AisleMode.IDLE;
			
        END_IF

    E_AisleMode.FAULT:
        bBoxAtPickPoint    := FALSE;
        bReadyForRetrieval := FALSE;
        bError             := TRUE;

END_CASE

IF iAisleBelt.bError THEN
    eMode := E_AisleMode.FAULT;
END_IF

ACTION ACT_ConfigureAisle:
IF nAisleNumber = 1 THEN
    bEntrySensor  := GVL_IO.bAisle1EntrySensor;
    bCraneStation := GVL_IO.bAisle1CraneStation;
    GVL_IO.bAisle1MotorForward := iAisleBelt.bMotorRun AND NOT iAisleBelt.bMotorReverse;
    GVL_IO.bAisle1MotorReverse := iAisleBelt.bMotorRun AND iAisleBelt.bMotorReverse;
ELSE
    bEntrySensor  := GVL_IO.bAisle2EntrySensor;
    bCraneStation := GVL_IO.bAisle2CraneStation;
    GVL_IO.bAisle2MotorForward := iAisleBelt.bMotorRun AND NOT iAisleBelt.bMotorReverse;
    GVL_IO.bAisle2MotorReverse := iAisleBelt.bMotorRun AND iAisleBelt.bMotorReverse;
END_IF
END_ACTION

END_FUNCTION_BLOCK

// ---- POUs/Controller/FB_CraneController.TcPOU
FUNCTION_BLOCK FB_CraneController
VAR_INPUT
    nAisleNumber    : INT;
	iCrane          : I_Crane;
END_VAR
VAR_OUTPUT
    bBusy           : BOOL;
    bError          : BOOL;
   
END_VAR

VAR
	stCraneJob      : ST_CraneJob;
    stAisleStation  : ST_Position;
    stRackTarget    : ST_Position;
    bJobPending     : BOOL;
    bIsStore        : BOOL;
    nState          : (IDLE, DISPATCHING, EXECUTING, DONE) := IDLE;
	stEmptySlot : ST_StorageSlot;
END_VAR


bBusy  := iCrane.bBusy;
bError := iCrane.bError;

CASE nState OF

    IDLE:
       
        IF bJobPending THEN
            nState := DISPATCHING;
        END_IF

    DISPATCHING:
        stAisleStation.fTargetX        := GVL_Config.HOME_X;
        stAisleStation.fTargetY        := GVL_Config.HOME_Y;
        stAisleStation.bIsAisleStation := TRUE;
        IF bIsStore THEN
            iCrane.M_StartJob(stPick := stAisleStation, stPlace := stRackTarget);
        ELSE
            iCrane.M_StartJob(stPick := stRackTarget, stPlace := stAisleStation);
        END_IF
        bJobPending := FALSE;
        nState      := EXECUTING;

    EXECUTING:
    IF iCrane.eState = E_CraneState.IDLE THEN

        IF stCraneJob.bIsStore THEN
            GVL_Warehouse.arrRack[stCraneJob.stRackPos.nRow, stCraneJob.stRackPos.nCol].eStatus := E_SlotStatus.OCCUPIED;
			GVL_Warehouse.nTotalStoredCount := GVL_Warehouse.nTotalStoredCount + 1;
        ELSE
            GVL_Warehouse.arrRack[stCraneJob.stRackPos.nRow, stCraneJob.stRackPos.nCol].eStatus := E_SlotStatus.EMPTY;     
			GVL_Warehouse.arrRack[stCraneJob.stRackPos.nRow, stCraneJob.stRackPos.nCol].stParcel := stEmptySlot.stParcel;     
			GVL_Warehouse.nTotalRetrievedCount := GVL_Warehouse.nTotalRetrievedCount + 1;
            
        END_IF
        nState := DONE;
    END_IF

    DONE:
        nState    := IDLE;

END_CASE

IF iCrane.bError THEN
    bJobPending := FALSE;
    nState      := IDLE;
END_IF

METHOD M_AssignRetrieve : BOOL
VAR_INPUT
   stJob : ST_CraneJob;
END_VAR
IF nState <> IDLE OR bJobPending THEN
    M_AssignRetrieve := FALSE;
    RETURN;
END_IF
stCraneJob := stJob;
stRackTarget  := stJob.stRackPos;
bIsStore         := FALSE;
bJobPending      := TRUE;
M_AssignRetrieve := TRUE;
END_METHOD

METHOD M_AssignStore : BOOL
VAR_INPUT
    stJob : ST_CraneJob;
END_VAR
IF nState <> IDLE OR bJobPending THEN
    M_AssignStore := FALSE;
    RETURN;
END_IF
stCraneJob := stJob;
stRackTarget  := stJob.stRackPos;
bIsStore      := TRUE;
bJobPending   := TRUE;
M_AssignStore := TRUE;
END_METHOD

END_FUNCTION_BLOCK

// ---- POUs/Controller/FB_OutFeedController.TcPOU
FUNCTION_BLOCK FB_OutFeedController
VAR_OUTPUT
    bBusy           : BOOL;
    bError          : BOOL;
    bComplete       : BOOL;
	
END_VAR
VAR
    nState : (IDLE, RUNNING, DONE) := IDLE;
END_VAR
VAR_INPUT
	iOutfeedBelt    : I_Conveyor;
END_VAR

GVL_IO.bOutfeedMotor := iOutfeedBelt.bMotorRun;

CASE nState OF

    IDLE:
        bBusy     := FALSE;
        bComplete := FALSE;
        
        IF GVL_IO.bOutfeedApproachSensor AND NOT GVL_IO.bOutfeedExitSensor THEN
			GVL_IO.bOutfeedStopBlocker := TRUE;
            iOutfeedBelt.M_Run(bForward := TRUE);
            bBusy  := TRUE;
            nState := RUNNING;
        END_IF

    RUNNING:
       
        IF GVL_IO.bOutfeedExitSensor THEN
			GVL_IO.bOutfeedApproachSensor := FALSE;
			GVL_IO.bOutfeedReq := FALSE;
            iOutfeedBelt.M_Stop();
            bComplete := TRUE;
            nState    := DONE;
        END_IF

    DONE:
        bBusy  := FALSE;
        nState := IDLE;

END_CASE

bError := iOutfeedBelt.bError;

END_FUNCTION_BLOCK
